PROGRAM MAIN_OLD
VAR
	// Linear wave parameters, Hs = 8 and Tp = 12.0;
	w0 AT %Q* : LREAL := 0.5457;
	lambda AT %Q* : LREAL := 0.2405;
	sigma AT %Q* : LREAL := 1.5012;
	
	// HMI data
	txHmi : ST_TxHmi;
	rxHmi : ST_RxHmi;
	
	// HMI activity check
	hmiCounterOld : UDINT := 0;
	hmiTimer : TON;
	
	// Remote interface
	//remote : FB_RemoteInterface('192.168.90.60', 50060, 50050);
	
	// Machinery
	em8000 : FB_StewartInterface('192.168.90.30', 50030, 50040, ADR(txHmi.em8000));
	em1500 : FB_StewartInterface('192.168.90.31', 50031, 50041, ADR(txHmi.em1500));
	comau : FB_ComauInterface('192.168.90.32', 50032, 50042, ADR(txHmi.comau));
	winch : FB_WinchInterface(ADR(txHmi.winch));
	
	// Sensors
	mru1 : FB_MruInterface(50043, ADR(txHmi.mru1));
	mru2 : FB_MruInterface(50044, ADR(txHmi.mru2));
	qtm : FB_QualisysInterface(50199, ADR(txHmi.qtm));
	at960 : FB_LeicaInterface;
	
	// Timing
	t : LREAL := 0.0;
	Ts : LREAL := 0.005;
	
	// Contorl and Feedback structs
	control : ST_Control;
	feedback : ST_Feedback;
	
	// Trajectory Speed seetings
	qDotMax : LREAL := 10.0/180.0*PI; // rad/s
	lengthDotMax : LREAL := 0.3; // m/s
	
	// EKF Estimator
	init : SINT := 0;
	pendelEstimator : FB_PendelEstimator;
	
	// LQR Anti Swing Controller
	lqrAntiSwing : FB_LqrAntiSwing;
	
	// Control Mapping
	controlMapping : FB_ControlMapping;

	// Winch Contorller
	winchController : FB_WinchController;
	length : LREAL;
	lengthOld : LREAL;
	lengthDot : LREAL;
	
	// System call for starting PqQt HMI
	fbStartProcess : NT_StartProcess;
	
	phi : ARRAY [0..1] OF LREAL;
END_VAR


// Update sensors and equipement
em8000();
em1500();
mru1();
mru2();
at960();
qtm();





// Feedback Struct
feedback.em8000 := em8000.feedback;
feedback.em1500 := em1500.feedback;
feedback.comau := comau.feedback;
feedback.at960 := at960.feedback;
feedback.mru1 := mru1.feedback;
feedback.mru2 := mru2.feedback;
feedback.winch := winch.feedback;
feedback.qtm := qtm.feedback;

// Control Struct
control.em8000 := em8000.control;
control.em1500 := em1500.control;
control.comau := comau.control;
control.winch := winch.control;

// Winch Controller
winchController(
	lengthExtra := LIMIT(-2.5, winchController.lengthExtra - lengthDotMax*rxHmi.xboxRightY*Ts, -0.841),
	lengthExtra_t := - lengthDotMax*rxHmi.xboxRightY*Ts,
	stFeedback := feedback
);

length := winchController.stWinchControl.length;
lengthDot := (length - lengthOld)/Ts;
lengthOld := length;

// EKF Estimator
IF qtm.active THEN
	pendelEstimator(
		Ts := Ts,
		stFeedback := feedback
	);
ELSE
	pendelEstimator(
		Ts := Ts,
		reset := TRUE,
		stFeedback := feedback
	);
END_IF
	
// Return estimator values to HMI
txHmi.phi[0] := LREAL_TO_REAL(pendelEstimator.phi[0]);
txHmi.phi[1] := LREAL_TO_REAL(pendelEstimator.phi[1]);

txHmi.phi_t[0] := LREAL_TO_REAL(pendelEstimator.phi_t[0]);
txHmi.phi_t[1] := LREAL_TO_REAL(pendelEstimator.phi_t[1]);

txHmi.e[0] := LREAL_TO_REAL(pendelEstimator.e[0]);
txHmi.e[1] := LREAL_TO_REAL(pendelEstimator.e[1]);
txHmi.e[2] := LREAL_TO_REAL(pendelEstimator.e[2]);

txHmi.c := LREAL_TO_REAL(pendelEstimator.c);

(*
// Anti Swing Controller
lqrAntiSwing(
	Ts := Ts,
	LQRmAX := 0.5,
	phi := pendelEstimator.phi,
	phi_t := pendelEstimator.phi_t
);

// Control Mapping
controlMapping.p := lqrAntiSwing.p;
controlMapping.p_t := lqrAntiSwing.p_t;

controlMapping.q0[0] := LIMIT(-25.0/180.0*PI, controlMapping.q0[0] + (rxHmi.xboxRT - rxHmi.xboxLT)*qDotMax*Ts, 35.0/180.0*PI);
controlMapping.q0_t[0] := (rxHmi.xboxRT - rxHmi.xboxLT)*qDotMax;

controlMapping.q0[1] := LIMIT(-10.0/180.0*PI, controlMapping.q0[1] + rxHmi.xboxLeftX*qDotMax*Ts, 15.0/180.0*PI);
controlMapping.q0_t[1] := rxHmi.xboxLeftX*qDotMax;

//controlMapping.q0[2] := LIMIT(-110.0/180.0*PI, controlMapping.q0[2] + rxHmi.xboxLeftY*qDotMax*Ts, -90.0/180.0*PI);
//controlMapping.q0_t[2] := rxHmi.xboxLeftY*qDotMax;

controlMapping.q0[2] := -110.0/180.0*PI;


controlMapping(
	stFeedback := feedback
);



// Apply contollers
winch.control.length := length;
winch.control.length_t := lengthDot;

comau.control := controlMapping.stControlComau;
*)


// Update elements to be controlled
comau();
winch();

t := t + Ts;


// Auto after given time without HMI activity
hmiTimer.PT := T#2S;

IF rxHmi.counter <> hmiCounterOld THEN
	hmiCounterOld := rxHmi.counter;
	hmiTimer.IN := TRUE;
ELSE
	hmiTimer.IN := FALSE;
END_IF

IF hmiTimer.Q THEN
	// Shutdown procedure here...
	
END_IF

ACTION StartPyQtHMI:
fbStartProcess(
	NETID := '192.168.90.160.1.1',
	PATHSTR := 'C:\motion-lab\hmi\startHMI.bat',
	DIRNAME := 'C:\motion-lab\hmi',
	COMNDLINE := 'startHMI.bat',
	START := TRUE
);
END_ACTION

END_PROGRAM

(* stored: Version 1.1.0.1, ProductVersion 3.1.4022.18
   POU MAIN_OLD: Id {4193d1f4-5b8a-4d46-8bb1-f5443e3607b6}, SpecialFunc None
   Action StartPyQtHMI: Id {9bb8c736-3772-4a32-953f-a2d6b917a904} *)
